// TIA Portal V18 export
// export: Created 2025-12-01T17:53:08.3655575Z, ExportSetting None, DisplayName Totally Integrated Automation Portal, DisplayVersion V18 Update 5, DisplayName TIA Portal Openness, DisplayVersion V18 Update 5, DisplayName TIA Portal Teamcenter Gateway, DisplayVersion V18, DisplayName TIA Portal Version Control Interface, DisplayVersion V18, DisplayName STEP 7 Professional, DisplayVersion V18 Update 5, DisplayName STEP 7 Safety, DisplayVersion V18, DisplayName WinCC Professional, DisplayVersion V18 Update 5
Screen "710 Recipe"  1280x800, Number=710, Template=07Parameter
  ScreenLayer "Layer_0"
    Button "btnMenu3" at 256,725 size 128x75  StyleItem=BtnNormal20, TextOff="Text", TextOn="Text"
    Button "btnMenu4" at 384,725 size 128x75  StyleItem=BtnNormal20, TextOff="Text", TextOn="Text"
    Button "btnMenu5" at 512,725 size 128x75  StyleItem=BtnNormal20, TextOff="Text", TextOn="Text"
    Button "btnMenu6" at 768,725 size 128x75  StyleItem=BtnNormal20, TextOff="Text", TextOn="Text"
    Button "btnMenu5_1" at 640,725 size 128x75  StyleItem=BtnNormal20, TextOff="Text", TextOn="Text"
    Button "btnMenu6_1" at 896,725 size 128x75  StyleItem=BtnNormal20, TextOff="Text", TextOn="Text"
    Button "btnMenu3_1" at 128,725 size 128x75  StyleItem=BtnNormal20, TextOff="Text", TextOn="Text"
    Button "btnMenu6_2" at 1152,725 size 128x75  StyleItem=BtnNormal20, TextOff="Text", TextOn="Text"
